// TIA Portal V17 export
// export: Created 2022-07-28T18:02:44.7250723Z, ExportSetting None, DisplayName Totally Integrated Automation Portal, DisplayVersion V17, DisplayName TIA Portal Openness, DisplayVersion V17, DisplayName TIA Portal Teamcenter Gateway, DisplayVersion V17, DisplayName TIA Portal Version Control Interface, DisplayVersion V17, DisplayName TIA Portal Test Suite Advanced, DisplayVersion V17, DisplayName SINAMICS Startdrive Advanced, DisplayVersion V17, DisplayName SINAMICS DCC, DisplayVersion V17, DisplayName SINAMICS Startdrive G130, G150, S120, S150, SINAMICS MV, S210, DisplayVersion V17, DisplayName SINAMICS Startdrive G110M, G120, G120C, G120D, G120P, G115D, DisplayVersion V17, DisplayName STEP 7 Professional, DisplayVersion V17, DisplayName SIMATIC Energy Suite, DisplayVersion V17, DisplayName STEP 7 CFC, DisplayVersion V17, DisplayName STEP 7 Safety, DisplayVersion V17, DisplayName WinCC Advanced / Unified PC, DisplayVersion V17, DisplayName SIMATIC Visualization Architect, DisplayVersion V17
FUNCTION_BLOCK "Lib_FB_MotSimp"   // FB10, SCL
{ S7_Optimized_Access := 'TRUE' }
// stored: MemoryReserve 100, SetENOAutomatically false
   VAR_INPUT
      i_StartFwd : Bool;   // Start motor forward command
      i_StartRev : Bool;   // Start motor backward command
      i_FdbckFwd : Bool;   // Feedback forward
      i_FdbckRev : Bool;   // Feedback backward
      i_RestartingPLC : Bool;   // PLC restart is active
      i_SimMode : Bool;   // Simulation mode is active
      ir_TimeCycle : Real;   // PLC one cycle time, sec
      ir_SPTimeFdbck : Real;   // Setpoint for feedback fault detection, sec
      ir_SPTimeRev : Real;   // Delay before changing the direction of rotation, sec.
      ir_SPTimeNxtStrt : Real;   // Delay before next start, sec
   END_VAR
   VAR_OUTPUT
      q_CmdRunFwd : Bool;   // Start motor forward command
      q_CmdRunRev : Bool;   // Start motor backward command
      q_Fault : Bool;   // Some fault is ative
      qs_Statuses : Struct   // Motor statuses
         Run : Bool;   // Motor is running (any direction)
         RunFwd : Bool;   // Motor is running forward
         RunRev : Bool;   // Motor is running backward
         SimMode : Bool;   // Simulation mode is active
         AfterStpBlck : Bool;   // Delay (block) after motor stop
         CngDirBlck : Bool;   // Delay before direction changing
         ST_7 : Bool;   // Status #7
         ST_8 : Bool;   // Status #8
         FltStartFwdBwdActive : Bool;   // Start commands forward and backward are active
         FltFwdContOn : Bool;   // Fault of forward contactor start
         FltFwdContOff : Bool;   // Fault of forward contactor stop
         FltRevContOn : Bool;   // Fault of backward contactor start
         FltRevContOff : Bool;   // Fault of backward contactor stop
         FLT_6 : Bool;   // Fault #6
         FLT_7 : Bool;   // Fault #7
         FLT_8 : Bool;   // Fault #8
      END_STRUCT;
   END_VAR
   VAR
      s_CmdRunFwd { ExternalAccessible := 'False'; ExternalVisible := 'False'; ExternalWritable := 'False'} : Bool;   // Start motor forward command
      s_CmdRunBwd { ExternalAccessible := 'False'; ExternalVisible := 'False'; ExternalWritable := 'False'} : Bool;   // Start motor backward command
      s_OldDirFwd { ExternalAccessible := 'False'; ExternalVisible := 'False'; ExternalWritable := 'False'} : Bool := true;   // Last direction (true = forward)
      sfb_TOF_ChngDir { ExternalAccessible := 'False'; ExternalVisible := 'False'; ExternalWritable := 'False'} : "Lib_FB_Timer_OFF_Simple";   // Changing the direction of rotation timer
      sfb_TOF_NxtStrt { ExternalAccessible := 'False'; ExternalVisible := 'False'; ExternalWritable := 'False'} : "Lib_FB_Timer_OFF_Simple";   // Deley beetween motor starts
      sfb_TON_FwdFdbck { ExternalAccessible := 'False'; ExternalVisible := 'False'; ExternalWritable := 'False'} : "Lib_FB_Timer_ON_Simple";   // Feedback from contactor on (forward)
      sfb_TON_BwdFdbck { ExternalAccessible := 'False'; ExternalVisible := 'False'; ExternalWritable := 'False'} : "Lib_FB_Timer_ON_Simple";   // Feedback from contactor on (backward)
   END_VAR
   VAR_TEMP
      t_StrtFwdPermtd : Bool;   // Start forward is permited
      t_StrtBwdPermtd : Bool;   // Start backward is permited
      t_FwdContFdbck : Bool;   // Forward contactor feedback (standard and sim mode)
      t_BwdContFdbck : Bool;   // Backward contactor feedback (standard and sim mode)
      t_SomeFault : Bool;   // Some fault is active
      t_FwdContOnFlt : Bool;   // Fault of forward contactor start
      t_FwdContOffFlt : Bool;   // Fault of forward contactor stop
      t_BwdContOnFlt : Bool;   // Fault of backward contactor start
      t_BwdContOffFlt : Bool;   // Fault of backward contactor stop
      t_CngDirFwdBlck : Bool;   // Delay before direction changing
      t_CngDirBwdBlck : Bool;   // Delay before direction changing
      t_NxtStrtBlck : Bool;   // Next start block
   END_VAR
BEGIN
   REGION Description
       //   Блок керування контактором мотора
       //   Входи iStartFwd та iStartRev ініціалізує запуск контактора руху мотора вперед і назад відповідно.
       //   Якщо після подачі команди iStartFwd на входах блоку не з'являється сигнал зворотнього зв'язку iFdbckFwd впродорвж часу irSPTimeFdbck (сек), то помилка запуску контактора osStatuses.FltFwdContOn стає активною. Вона буде активною, поки команда iStartFwd не стане рівною 0.
       //   Після того, як сигнал про запуск iStartFwd зникає, а сигнал зворотнього зв'язку iFdbckFwd впродорвж часу irSPTimeFdbck не зникає, то помилка зупинки контактора osStatuses.FltFwdContOff стає активною.
       //   Блок керування контактором мотора
       //   Аналогічна логіка і для контактора руху мотора назад.
       //   При появі одночасно сигналів iStartFwd та iStartRev, активується аварія osStatuses.FltStartFwdBwdActive.
       //   При появі будь-якої з перелічених помилок, подача сигналу 'Пуск' на контактори припиняється.
       //   Крім того існують блокування, які захищають пускачі від частих стартів і від ввімкнення двигуна у протифазі. Інтервали часу, впродовж яких ці блокування активні, задаються на входах irSPTimeNxtStrt та irSPTimeRev відповідно. Відлік часу починається з моменту припинення подачі команди 'Пуск' на пускач.
       //   Симулювати роботу блоку можна, якщо подати на вхід iSimMode сигнал true. В такому режимі, при подачі сигналу запуску, симулюється відповідний зворотній зв'язок контактора, але команди запуску не подаються на виходи oCmdRunFwd та oCmdRunRev, а лише відображаються в структурі osStatuses.   

       //   Motor contactor control unit
       //   The iStartFwd and iStartRev inputs initiate the start of the forward and reverse motor contactor, respectively.
       //   If the iFtbckFwd feedback signal does not appear on the inputs of the block after the iStartFwd command is issued during the irSPTimeFdbck time (sec), the error of starting the contactor osStatuses.FltFwdContOn becomes active. It will remain active until the iStartFwd command becomes 0.
       //   After the iStartFwd start signal disappears and the iFdbckFwd feedback signal does not disappear during the irSPTimeFdbck time, the stop error of the osStatuses.FltFwdContOff contactor becomes active.
       //   The logic is similar for the contactor of the motor movement back.
       //   If the iStartFwd and iStartRev signals appear at the same time, the osStatuses.FltStartFwdBwdActive alarm is activated.
       //   If any of these errors occur, the 'Start' signal to the contactors is stopped.
       //   In addition, there are locks that protect the contactors from frequent starts and from starting the motor in antiphase. The time intervals during which these locks are active are set on the irSPTimeNxtStrt and irSPTimeRev inputs, respectively. The countdown starts from the moment the command "Start" on the contactor is stopped.
       //   You can simulate the operation of the unit if you send a true signal to the iSimMode input. In this mode, when the start signal is applied, the corresponding feedback of the contactor is simulated, but the start commands are not given to the outputs oCmdRunFwd and oCmdRunRev, but are only displayed in the osStatuses structure.    
   END_REGION

   REGION Feedback signal (standard and sim mode)
       #t_FwdContFdbck := #i_FdbckFwd OR (#s_CmdRunFwd AND #i_SimMode);    //Forward contactor feedback (standard and sim mode)
       #t_BwdContFdbck := #i_FdbckRev OR (#s_CmdRunBwd AND #i_SimMode);    //Backward contactor feedback (standard and sim mode)
   END_REGION

   REGION Timers
       REGION Timers setpoints
           #sfb_TOF_ChngDir.IR_SpTime := #ir_SPTimeRev; //Changing the direction of rotation timer

           #sfb_TOF_NxtStrt.IR_SpTime := #ir_SPTimeNxtStrt; //Deley beetween motor starts

           #sfb_TON_FwdFdbck.IR_SpTime := #ir_SPTimeFdbck;  //Feedback from contactor on (forward)
           #sfb_TON_BwdFdbck.IR_SpTime := #ir_SPTimeFdbck;  //Feedback from contactor on (backward)
       END_REGION

       REGION Timers inputsts
           #sfb_TOF_ChngDir.IB_StartTimerInput := #s_CmdRunFwd  //Changing the direction of rotation timer
           OR #s_CmdRunBwd
           ;

           #sfb_TOF_NxtStrt.IB_StartTimerInput := #s_CmdRunFwd  //Deley beetween motor starts
           OR #s_CmdRunBwd
           OR #i_FdbckFwd
           OR #i_FdbckRev
           ;

           #sfb_TON_FwdFdbck.IB_StartTimerInput := (#s_CmdRunFwd    //Feedback from contactor on (forward)
           AND NOT #t_FwdContFdbck)

           OR (#sfb_TON_FwdFdbck.QB_TimerOut
           AND NOT #t_FwdContFdbck
           AND #i_StartFwd)

           OR (NOT #s_CmdRunFwd
           AND #t_FwdContFdbck)

           OR (#sfb_TON_FwdFdbck.QB_TimerOut
           AND #t_FwdContFdbck
           AND NOT #i_StartFwd)
           ;

           #sfb_TON_BwdFdbck.IB_StartTimerInput := (#s_CmdRunBwd    //Feedback from contactor on (backward)
           AND NOT #t_BwdContFdbck)

           OR (#sfb_TON_BwdFdbck.QB_TimerOut
           AND NOT #t_BwdContFdbck
           AND #i_StartRev)

           OR (NOT #s_CmdRunBwd
           AND #t_BwdContFdbck)

           OR (#sfb_TON_BwdFdbck.QB_TimerOut
           AND #t_BwdContFdbck
           AND NOT #i_StartRev)
           ;
       END_REGION

       REGION Timers calling 
           //PLC cycle time
           #sfb_TOF_ChngDir.IR_CycleTime :=        //Changing the direction of rotation timer
           #sfb_TOF_NxtStrt.IR_CycleTime :=        //Deley beetween motor starts
           #sfb_TON_FwdFdbck.IR_CycleTime :=       //Feedback from contactor on (forward)
           #sfb_TON_BwdFdbck.IR_CycleTime :=       //Feedback from contactor on (backward)
           #ir_TimeCycle;
           //Timers functions
           #sfb_TOF_ChngDir();     //Changing the direction of rotation timer
           #sfb_TOF_NxtStrt();     //Deley beetween motor starts
           #sfb_TON_FwdFdbck();    //Feedback from contactor on (forward)
           #sfb_TON_BwdFdbck();    //Feedback from contactor on (backward)
       END_REGION
   END_REGION

   REGION Old direction
       //Last direction (true = forward)
       IF #s_CmdRunFwd THEN
           #s_OldDirFwd := 1;
       ELSIF #s_CmdRunBwd THEN
           #s_OldDirFwd := 0;
       END_IF;
   END_REGION

   REGION Block start/stop
       //Delay before direction changing
       #t_CngDirFwdBlck := (#sfb_TOF_ChngDir.QB_TimerOut AND NOT #s_CmdRunFwd)
       AND NOT #s_OldDirFwd
       ;
       //Delay before direction changing
       #t_CngDirBwdBlck := (#sfb_TOF_ChngDir.QB_TimerOut AND NOT #s_CmdRunBwd)
       AND #s_OldDirFwd
       ;
       //Next start block
       #t_NxtStrtBlck := #sfb_TOF_NxtStrt.QB_TimerOut
       AND NOT (#s_CmdRunFwd
       OR #s_CmdRunBwd
       OR #i_FdbckFwd
       OR #i_FdbckRev)
       ;
   END_REGION

   REGION Faults
       #t_FwdContOnFlt := #sfb_TON_FwdFdbck.QB_TimerOut AND NOT #t_FwdContFdbck; //Fault of forward contactor start
       #t_BwdContOnFlt := #sfb_TON_BwdFdbck.QB_TimerOut AND NOT #t_BwdContFdbck; //Fault of backward contactor start

       #t_FwdContOffFlt := #sfb_TON_FwdFdbck.QB_TimerOut AND #t_FwdContFdbck;    //Fault of forward contactor stop
       #t_BwdContOffFlt := #sfb_TON_BwdFdbck.QB_TimerOut AND #t_BwdContFdbck;    //Fault of backward contactor stop

       //Some fault is active
       #t_SomeFault := #t_FwdContOnFlt
       OR #t_BwdContOnFlt
       OR #t_FwdContOffFlt
       OR #t_BwdContOffFlt
       OR (#i_StartFwd AND #i_StartRev)
       ;
   END_REGION

   REGION Start permitions
       //Start forward is permited
       #t_StrtFwdPermtd := NOT #t_CngDirFwdBlck
       AND NOT #t_NxtStrtBlck
       AND NOT #t_SomeFault
       ;
       //Start backward is permited
       #t_StrtBwdPermtd := NOT #t_CngDirBwdBlck
       AND NOT #t_NxtStrtBlck
       AND NOT #t_SomeFault
       ;
       REGION Description
           //   Блок керування контактором мотора
           //   Входи iStartFwd та iStartRev ініціалізує запуск контактора руху мотора вперед і назад відповідно.
           //   Якщо після подачі команди iStartFwd на входах блоку не з'являється сигнал зворотнього зв'язку iFdbckFwd впродорвж часу irSPTimeFdbck (сек), то помилка запуску контактора osStatuses.FltFwdContOn стає активною. Вона буде активною, поки команда iStartFwd не стане рівною 0.
           //   Після того, як сигнал про запуск iStartFwd зникає, а сигнал зворотнього зв'язку iFdbckFwd впродорвж часу irSPTimeFdbck не зникає, то помилка зупинки контактора osStatuses.FltFwdContOff стає активною.
           //   Блок керування контактором мотора
           //   Аналогічна логіка і для контактора руху мотора назад.
           //   При появі одночасно сигналів iStartFwd та iStartRev, активується аварія osStatuses.FltStartFwdBwdActive.
           //   При появі будь-якої з перелічених помилок, подача сигналу 'Пуск' на контактори припиняється.
           //   Крім того існують блокування, які захищають пускачі від частих стартів і від ввімкнення двигуна у протифазі. Інтервали часу, впродовж яких ці блокування активні, задаються на входах irSPTimeNxtStrt та irSPTimeRev відповідно. Відлік часу починається з моменту припинення подачі команди 'Пуск' на пускач.
           //   Симулювати роботу блоку можна, якщо подати на вхід iSimMode сигнал true. В такому режимі, при подачі сигналу запуску, симулюється відповідний зворотній зв'язок контактора, але команди запуску не подаються на виходи oCmdRunFwd та oCmdRunRev, а лише відображаються в структурі osStatuses.   

           //   Motor contactor control unit
           //   The iStartFwd and iStartRev inputs initiate the start of the forward and reverse motor contactor, respectively.
           //   If the iFtbckFwd feedback signal does not appear on the inputs of the block after the iStartFwd command is issued during the irSPTimeFdbck time (sec), the error of starting the contactor osStatuses.FltFwdContOn becomes active. It will remain active until the iStartFwd command becomes 0.
           //   After the iStartFwd start signal disappears and the iFdbckFwd feedback signal does not disappear during the irSPTimeFdbck time, the stop error of the osStatuses.FltFwdContOff contactor becomes active.
           //   The logic is similar for the contactor of the motor movement back.
           //   If the iStartFwd and iStartRev signals appear at the same time, the osStatuses.FltStartFwdBwdActive alarm is activated.
           //   If any of these errors occur, the 'Start' signal to the contactors is stopped.
           //   In addition, there are locks that protect the contactors from frequent starts and from starting the motor in antiphase. The time intervals during which these locks are active are set on the irSPTimeNxtStrt and irSPTimeRev inputs, respectively. The countdown starts from the moment the command "Start" on the contactor is stopped.
           //   You can simulate the operation of the unit if you send a true signal to the iSimMode input. In this mode, when the start signal is applied, the corresponding feedback of the contactor is simulated, but the start commands are not given to the outputs oCmdRunFwd and oCmdRunRev, but are only displayed in the osStatuses structure.    
       END_REGION

       REGION Feedback signal (standard and sim mode)
           #t_FwdContFdbck := #i_FdbckFwd OR (#s_CmdRunFwd AND #i_SimMode);    //Forward contactor feedback (standard and sim mode)
           #t_BwdContFdbck := #i_FdbckRev OR (#s_CmdRunBwd AND #i_SimMode);    //Backward contactor feedback (standard and sim mode)
       END_REGION

       REGION Timers
           REGION Timers setpoints
               #sfb_TOF_ChngDir.IR_SpTime := #ir_SPTimeRev; //Changing the direction of rotation timer

               #sfb_TOF_NxtStrt.IR_SpTime := #ir_SPTimeNxtStrt; //Deley beetween motor starts

               #sfb_TON_FwdFdbck.IR_SpTime := #ir_SPTimeFdbck;  //Feedback from contactor on (forward)
               #sfb_TON_BwdFdbck.IR_SpTime := #ir_SPTimeFdbck;  //Feedback from contactor on (backward)
           END_REGION

           REGION Timers inputsts
               #sfb_TOF_ChngDir.IB_StartTimerInput := #s_CmdRunFwd  //Changing the direction of rotation timer
               OR #s_CmdRunBwd
               ;

               #sfb_TOF_NxtStrt.IB_StartTimerInput := #s_CmdRunFwd  //Deley beetween motor starts
               OR #s_CmdRunBwd
               OR #i_FdbckFwd
               OR #i_FdbckRev
               ;

               #sfb_TON_FwdFdbck.IB_StartTimerInput := (#s_CmdRunFwd    //Feedback from contactor on (forward)
               AND NOT #t_FwdContFdbck)

               OR (#sfb_TON_FwdFdbck.QB_TimerOut
               AND NOT #t_FwdContFdbck
               AND #i_StartFwd)

               OR (NOT #s_CmdRunFwd
               AND #t_FwdContFdbck)

               OR (#sfb_TON_FwdFdbck.QB_TimerOut
               AND #t_FwdContFdbck
               AND NOT #i_StartFwd)
               ;

               #sfb_TON_BwdFdbck.IB_StartTimerInput := (#s_CmdRunBwd    //Feedback from contactor on (backward)
               AND NOT #t_BwdContFdbck)

               OR (#sfb_TON_BwdFdbck.QB_TimerOut
               AND NOT #t_BwdContFdbck
               AND #i_StartRev)

               OR (NOT #s_CmdRunBwd
               AND #t_BwdContFdbck)

               OR (#sfb_TON_BwdFdbck.QB_TimerOut
               AND #t_BwdContFdbck
               AND NOT #i_StartRev)
               ;
           END_REGION

           REGION Timers calling 
               //PLC cycle time
               #sfb_TOF_ChngDir.IR_CycleTime :=        //Changing the direction of rotation timer
               #sfb_TOF_NxtStrt.IR_CycleTime :=        //Deley beetween motor starts
               #sfb_TON_FwdFdbck.IR_CycleTime :=       //Feedback from contactor on (forward)
               #sfb_TON_BwdFdbck.IR_CycleTime :=       //Feedback from contactor on (backward)
               #ir_TimeCycle;
               //Timers functions
               #sfb_TOF_ChngDir();     //Changing the direction of rotation timer
               #sfb_TOF_NxtStrt();     //Deley beetween motor starts
               #sfb_TON_FwdFdbck();    //Feedback from contactor on (forward)
               #sfb_TON_BwdFdbck();    //Feedback from contactor on (backward)
           END_REGION
       END_REGION

       REGION Old direction
           //Last direction (true = forward)
           IF #s_CmdRunFwd THEN
               #s_OldDirFwd := 1;
           ELSIF #s_CmdRunBwd THEN
               #s_OldDirFwd := 0;
           END_IF;
       END_REGION

       REGION Block start/stop
           //Delay before direction changing
           #t_CngDirFwdBlck := (#sfb_TOF_ChngDir.QB_TimerOut AND NOT #s_CmdRunFwd)
           AND NOT #s_OldDirFwd
           ;
           //Delay before direction changing
           #t_CngDirBwdBlck := (#sfb_TOF_ChngDir.QB_TimerOut AND NOT #s_CmdRunBwd)
           AND #s_OldDirFwd
           ;
           //Next start block
           #t_NxtStrtBlck := #sfb_TOF_NxtStrt.QB_TimerOut
           AND NOT (#s_CmdRunFwd
           OR #s_CmdRunBwd
           OR #i_FdbckFwd
           OR #i_FdbckRev)
           ;
       END_REGION

       REGION Faults
           #t_FwdContOnFlt := #sfb_TON_FwdFdbck.QB_TimerOut AND NOT #t_FwdContFdbck; //Fault of forward contactor start
           #t_BwdContOnFlt := #sfb_TON_BwdFdbck.QB_TimerOut AND NOT #t_BwdContFdbck; //Fault of backward contactor start

           #t_FwdContOffFlt := #sfb_TON_FwdFdbck.QB_TimerOut AND #t_FwdContFdbck;    //Fault of forward contactor stop
           #t_BwdContOffFlt := #sfb_TON_BwdFdbck.QB_TimerOut AND #t_BwdContFdbck;    //Fault of backward contactor stop

           //Some fault is active
           #t_SomeFault := #t_FwdContOnFlt
           OR #t_BwdContOnFlt
           OR #t_FwdContOffFlt
           OR #t_BwdContOffFlt
           OR (#i_StartFwd AND #i_StartRev)
           ;
       END_REGION

       REGION Start permitions
           //Start forward is permited
           #t_StrtFwdPermtd := NOT #t_CngDirFwdBlck
           AND NOT #t_NxtStrtBlck
           AND NOT #t_SomeFault
           ;
           //Start backward is permited
           #t_StrtBwdPermtd := NOT #t_CngDirBwdBlck
           AND NOT #t_NxtStrtBlck
           AND NOT #t_SomeFault
           ;
       END_REGION

       REGION Start commands
           //Start motor forward command
           #s_CmdRunFwd := #i_StartFwd
           AND NOT #i_StartRev
           AND #t_StrtFwdPermtd
           ;
           //Start motor backward command
           #s_CmdRunBwd := NOT #i_StartFwd
           AND #i_StartRev
           AND #t_StrtBwdPermtd
           ;
       END_REGION

       REGION Outputs
           #q_CmdRunFwd := #s_CmdRunFwd AND NOT #i_SimMode;   //Start motor forward command
           #q_CmdRunRev := #s_CmdRunBwd AND NOT #i_SimMode;   //Start motor backward command
           #q_Fault := #t_SomeFault;                         //Some fault is ative

           #qs_Statuses.Run := #t_FwdContFdbck OR #t_BwdContFdbck;    //Status Motor is running (any direction)
           #qs_Statuses.RunFwd := #t_FwdContFdbck;                    //Status Motor is running forward #s_CmdRunFwd AND 
           #qs_Statuses.RunRev := #t_BwdContFdbck;                    //Status Motor is running backward #s_CmdRunBwd AND 
           #qs_Statuses.SimMode := #i_SimMode;                       //Status Simulation mode is active
           #qs_Statuses.AfterStpBlck := #t_NxtStrtBlck               //Status Delay (block) after motor stop
           ;
           #qs_Statuses.CngDirBlck := (#t_CngDirFwdBlck              //Status Delay before direction changing
           AND #i_StartFwd)
           OR (#t_CngDirBwdBlck
           AND #i_StartRev)
           ;
           #qs_Statuses.FltStartFwdBwdActive := #i_StartFwd AND #i_StartRev;  //Fault Start forward and backward are active

           #qs_Statuses.FltFwdContOn := #t_FwdContOnFlt;             //Fault of forward contactor start 
           #qs_Statuses.FltFwdContOff := #t_FwdContOffFlt;           //Fault of forward contactor stop 
           #qs_Statuses.FltRevContOn := #t_BwdContOnFlt;             //Fault of backward contactor start 
           #qs_Statuses.FltRevContOff := #t_BwdContOffFlt;           //Fault of backward contactor stop 
       END_REGION

   END_REGION

   REGION Start commands
       //Start motor forward command
       #s_CmdRunFwd := #i_StartFwd
       AND NOT #i_StartRev
       AND #t_StrtFwdPermtd
       ;
       //Start motor backward command
       #s_CmdRunBwd := NOT #i_StartFwd
       AND #i_StartRev
       AND #t_StrtBwdPermtd
       ;
   END_REGION

   REGION Outputs
       #q_CmdRunFwd := #s_CmdRunFwd AND NOT #i_SimMode;   //Start motor forward command
       #q_CmdRunRev := #s_CmdRunBwd AND NOT #i_SimMode;   //Start motor backward command
       #q_Fault := #t_SomeFault;                         //Some fault is ative

       #qs_Statuses.Run := #t_FwdContFdbck OR #t_BwdContFdbck;    //Status Motor is running (any direction)
       #qs_Statuses.RunFwd := #t_FwdContFdbck;                    //Status Motor is running forward #s_CmdRunFwd AND 
       #qs_Statuses.RunRev := #t_BwdContFdbck;                    //Status Motor is running backward #s_CmdRunBwd AND 
       #qs_Statuses.SimMode := #i_SimMode;                       //Status Simulation mode is active
       #qs_Statuses.AfterStpBlck := #t_NxtStrtBlck               //Status Delay (block) after motor stop
       ;
       #qs_Statuses.CngDirBlck := (#t_CngDirFwdBlck              //Status Delay before direction changing
       AND #i_StartFwd)
       OR (#t_CngDirBwdBlck
       AND #i_StartRev)
       ;
       #qs_Statuses.FltStartFwdBwdActive := #i_StartFwd AND #i_StartRev;  //Fault Start forward and backward are active

       #qs_Statuses.FltFwdContOn := #t_FwdContOnFlt;             //Fault of forward contactor start 
       #qs_Statuses.FltFwdContOff := #t_FwdContOffFlt;           //Fault of forward contactor stop 
       #qs_Statuses.FltRevContOn := #t_BwdContOnFlt;             //Fault of backward contactor start 
       #qs_Statuses.FltRevContOff := #t_BwdContOffFlt;           //Fault of backward contactor stop 
   END_REGION
END_FUNCTION_BLOCK
